PROGRAM MAIN
VAR
	State: (INIT, OFF, ON, WARNING, ERROR); // {attribute 'to_string'}
	oState: STRING;
END_VAR

// ISSUE: Implicit/Private enum converts index instead of value when using TO_STRING
State := ON;
oState := TO_STRING(State); // EXP='OFF' ACT='2'

END_PROGRAM

(* stored: Version 1.1.0.1, ProductVersion 3.1.4024.11
   POU MAIN: Id {ed6cf280-cdd3-4860-bfde-a99a4c55cb3f}, SpecialFunc None *)
